Staubli VAL3: typeMenu.pgx

public program typeMenu(num pNumber, string pStr)
  local num lStep
  local num lPosY
  local string lStrEmpty
  local num lMaxLen
  local num i
  local string lStr
  local num lPosX
begin
  //---------------------------------
  //  S H O W   O N E   S T R I N G
  //---------------------------------
  // Display one message in the
  // user menu page
  // 4 characters and 1 space
  //
  //
  lStep=5
  lPosY=13
  lStrEmpty="     "
  if (pNumber>=1) and (pNumber<=8)
    lMaxLen=4
    // Control the len
    // europe case
    if (getDisplayLen(pStr)>lMaxLen)
      if len(pStr)==getDisplayLen(pStr)
        i=find(pStr," ")
        if i<5 and i>2
          lStr=mid(pStr,i,0)
        else
          lStr=mid(pStr,lMaxLen-1,0)
          lStr=lStr+"."
        endIf
      else
        // asia one
        lStr=mid(pStr,2,0)
      endIf
    else
      lStr=pStr
    endIf
    // Position X
    lPosX=(pNumber-1)*lStep+1
    // log
    call strfill(lStr,4,lStr)
    call type(lPosX,lPosY,lStr)
  endIf
end
